TYPE TcaTwinSAFEService :
STRUCT
	QuittButton : TcaPushButtonService;
	Safe : BOOL;
	Error : BOOL;
	Running : BOOL;
END_STRUCT
END_TYPE

(* stored: Version 1.1.0.1
   DUT TcaTwinSAFEService: Id {76179687-f2ce-429a-a7e9-ff251c7a7379} *)
